// TIA Portal V18 export
DATA_BLOCK "Mixing ratio"   // DB70
{ S7_Optimized_Access := 'TRUE' }
VERSION : 0.1
// stored: AutoNumber true, DBAccessibleFromOPCUA true, IsOnlyStoredInLoadMemory false, IsRetainMemResEnabled false, IsWriteProtectedInAS false, MemoryReserve 100
   VAR RETAIN
      "Mixing ratio according to density" : Real;
      "Mixing ratio set" : Real;
      "Mixing ratio tolerence for error" : Real;
      "Mixing ratio tolerence for warning" : Real;
   END_VAR
   VAR
      "Check MR" : Bool;
      "check mr0" : Bool;
      "Check MR ONS" : Bool;
      "Ratio check done" : Bool;
   END_VAR
   VAR RETAIN
      "MR check delay start time" : Int;
   END_VAR
   VAR
      "MR PV" : Real;
      "MR deviation" : Real;
      "Mixing ratio high Error" : Bool;
      "mixing ratio high Warning" : Bool;
      "Mixing ratio Low  Error" : Bool;
      "mixing ratio Low Warning" : Bool;
      "Mixing ratio Okay" : Bool;
      "Mixing ratio check done" : Bool;
      "mixing ratio check delay in Sec" : DInt;
      "ratio Min" : Real;
      "ratio max" : Real;
      "Mixing ratio Okay On recirculation" : Bool;
      "Mixing ratio error during recirculation" : Bool;
   END_VAR
BEGIN
END_DATA_BLOCK
